# EPICS autosave request: iocBoot/ioc13xps_smkb/auto_positions.req
file "CARS_motor_positions.req",         P=$(P), M=m1
file "CARS_motor_positions.req",         P=$(P), M=m2
file "CARS_motor_positions.req",         P=$(P), M=m3
file "CARS_motor_positions.req",         P=$(P), M=m4
file "CARS_motor_positions.req",         P=$(P), M=m5
